// TIA Portal V21 export
DATA_BLOCK "ModeDb"   // DB100
{ S7_Optimized_Access := 'FALSE' }
// stored: AutoNumber false
   VAR
      Cycle1 { S7_SetPoint := 'True'} : "ModePara";   // PHT
      Cycle2 { S7_SetPoint := 'True'} : "ModePara";   // BATCH
      Cycle3 { S7_SetPoint := 'True'} : "ModePara";   // SIP
      Cycle4 { S7_SetPoint := 'True'} : "ModePara";   // CIP
      Cycle5 { S7_SetPoint := 'True'} : "ModePara";   // LOAD CELL CALIBRATION
      VesselWeight { S7_SetPoint := 'True'} : Real;
      AlarmStarTime : DTL;
      AlarmEndTime : DTL;
   END_VAR
BEGIN
   Cycle2.CycleName := 'BATCH';
   Cycle3.CycleName := 'SIP';
   Cycle4.CycleName := 'CIP';
   Cycle5.CycleName := 'BULKSTRL';
END_DATA_BLOCK
